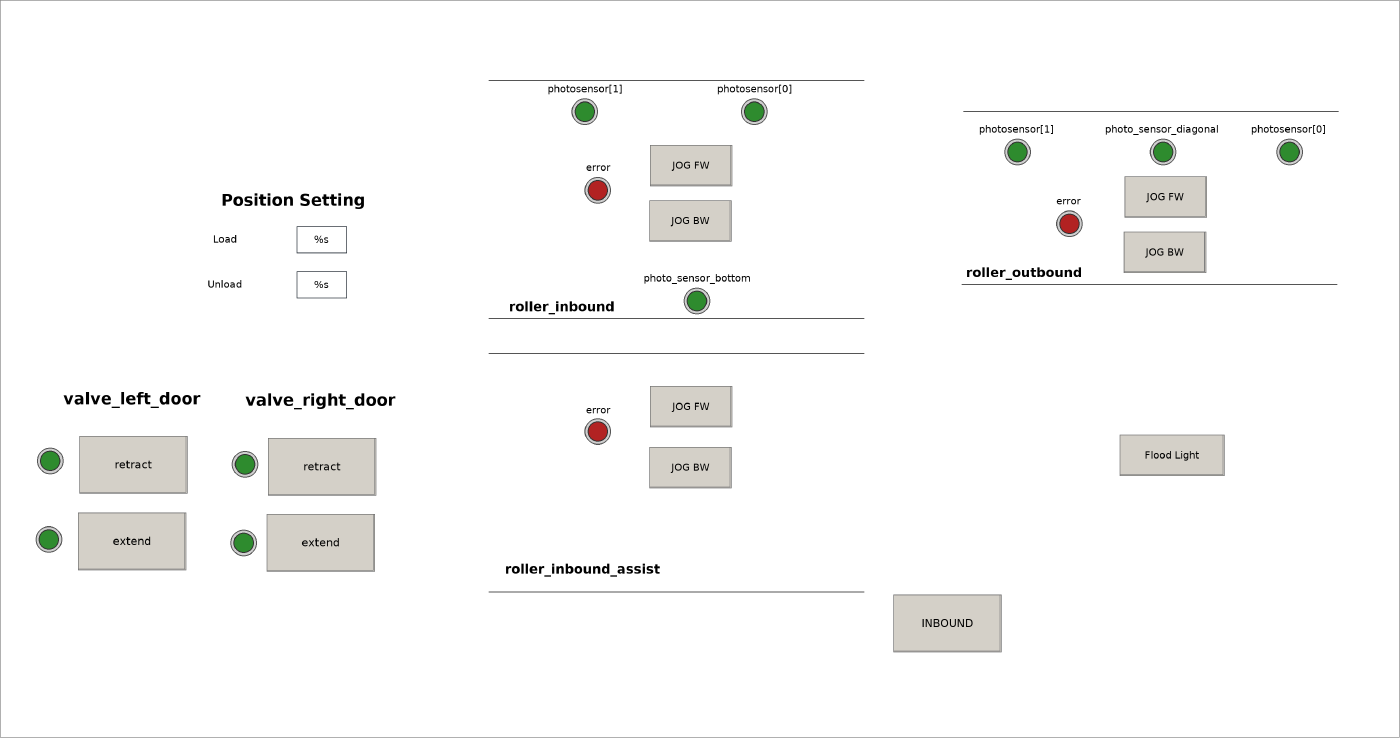
VISUALIZATION v_io_loading  // 2048x1080
    Lamp1 (1679,200 45x45), variable: GVL.fb_loading.photo_sensor_diagonal.Q, style: Lamp-Lamp1-Green
    Label (1600,176 200x26), "photo_sensor_diagonal"
    Lamp1 (1542,305 45x45), variable: GVL.fb_loading.roller_assign.roller.err.Q, style: Lamp-Lamp1-Red
    Label (1463,281 200x26), "error"
    Line (1409,163) (1958,163)
    Button (1645,258 120x60), "JOG FW", colour toggle: GVL.fb_loading.roller_assign.roller.forward
        OnMouseDown: execute { GVL.fb_loading.roller_assign.roller.forward	:= TRUE; }
        OnMouseUp: execute { GVL.fb_loading.roller_assign.roller.forward	:= FALSE; }
    Button (1644,339 120x60), "JOG BW", colour toggle: GVL.fb_loading.roller_assign.roller.backward
        OnMouseDown: execute { GVL.fb_loading.roller_assign.roller.backward	:= TRUE; }
        OnMouseUp: execute { GVL.fb_loading.roller_assign.roller.backward	:= FALSE; }
    Line (1407,416) (1956,416)
    Lamp1 (1864,200 45x45), variable: GVL.fb_loading.roller_assign.photo_sensor[0].Q, style: Lamp-Lamp1-Green
    Label (1785,176 200x26), "photosensor[0]"
    Lamp1 (1466,200 45x45), variable: GVL.fb_loading.roller_assign.photo_sensor[1].Q, style: Lamp-Lamp1-Green
    Label (1387,176 200x26), "photosensor[1]"
    Label (1398,384 200x30), "roller_outbound"
    Lamp1 (997,418 45x45), variable: GVL.fb_loading.photo_sensor_bottom.Q, style: Lamp-Lamp1-Green
    Label (920,394 200x26), "photo_sensor_bottom"
    Lamp1 (852,256 45x45), variable: GVL.fb_loading.roller_inbound.roller.err.Q, style: Lamp-Lamp1-Red
    Label (775,232 200x26), "error"
    Line (715,117) (1264,117)
    Button (951,212 120x60), "JOG FW", colour toggle: GVL.fb_loading.roller_inbound.roller.forward
        OnMouseDown: execute { GVL.fb_loading.roller_inbound.roller.forward	:= TRUE; }
        OnMouseUp: execute { GVL.fb_loading.roller_inbound.roller.forward	:= FALSE; }
    Button (950,293 120x60), "JOG BW", colour toggle: GVL.fb_loading.roller_inbound.roller.backward
        OnMouseDown: execute { GVL.fb_loading.roller_inbound.roller.backward	:= TRUE; }
        OnMouseUp: execute { GVL.fb_loading.roller_inbound.roller.backward	:= FALSE; }
    Line (715,466) (1264,466)
    Lamp1 (1081,141 45x45), variable: GVL.fb_loading.roller_inbound.photo_sensor[0].Q, style: Lamp-Lamp1-Green
    Label (1004,117 200x26), "photosensor[0]"
    Lamp1 (833,141 45x45), variable: GVL.fb_loading.roller_inbound.photo_sensor[1].Q, style: Lamp-Lamp1-Green
    Label (756,117 200x26), "photosensor[1]"
    Label (722,434 200x30), "roller_inbound"
    Button (1638,636 153x60), "Flood Light", colour toggle: GVL.fb_loading.floodlight
        toggle GVL.fb_loading.floodlight
        OnMouseDown: execute {  }
        OnMouseUp: execute {  }
    Rectangle (434,331 73x39), "%s", text variable: GVL.fb_loading.rPos_load
        OnMouseClick: write the text variable via Default, min GVL.fb_loading.rMin_lift, max GVL.fb_loading.rMax_lift
    Rectangle (434,397 73x39), "%s", text variable: GVL.fb_loading.rPos_unload
        OnMouseClick: write the text variable via Default, min GVL.fb_loading.rMin_lift, max GVL.fb_loading.rMax_lift
    Label (229,337 200x26), "Load"
    Label (229,403 200x26), "Unload"
    Label (254,280 350x26), "Position Setting"
    Lamp1 (852,609 45x45), variable: GVL.fb_loading.roller_inbound_assist.roller.err.Q, style: Lamp-Lamp1-Red
    Label (775,587 200x26), "error"
    Line (715,517) (1264,517)
    Button (951,565 120x60), "JOG FW", colour toggle: GVL.fb_loading.roller_inbound_assist.roller.forward
        OnMouseDown: execute { GVL.fb_loading.roller_inbound_assist.roller.forward	:= TRUE; }
        OnMouseUp: execute { GVL.fb_loading.roller_inbound_assist.roller.forward	:= false; }
    Button (950,654 120x60), "JOG BW", colour toggle: GVL.fb_loading.roller_inbound_assist.roller.backward
        OnMouseDown: execute { GVL.fb_loading.roller_inbound_assist.roller.backward 	:= TRUE; }
        OnMouseUp: execute { GVL.fb_loading.roller_inbound_assist.roller.backward	:= FALSE; }
    Line (715,866) (1264,866)
    Label (727,818 250x30), "roller_inbound_assist"
    Button (114,750 158x84), "extend", colour toggle: GVL.fb_loading.valve_left_door.extend
        OnMouseDown: execute { GVL.fb_loading.valve_left_door.retract := FALSE; GVL.fb_loading.valve_left_door.extend := TRUE; }
    Label (56,556 274x55), "valve_left_door"
    Button (116,638 158x84), "retract", colour toggle: GVL.fb_loading.valve_left_door.retract
        OnMouseDown: execute { GVL.fb_loading.valve_left_door.extend := FALSE; GVL.fb_loading.valve_left_door.retract := TRUE; }
    Button (390,752 158x84), "extend", colour toggle: GVL.fb_loading.valve_right_door.extend
        OnMouseDown: execute { GVL.fb_loading.valve_right_door.retract := FALSE; GVL.fb_loading.valve_right_door.extend := TRUE; }
    Label (332,558 274x55), "valve_right_door"
    Button (392,641 158x84), "retract", colour toggle: GVL.fb_loading.valve_right_door.retract
        OnMouseDown: execute { GVL.fb_loading.valve_right_door.extend := FALSE; GVL.fb_loading.valve_right_door.retract := TRUE; }
    Lamp1 (49,767 45x45), variable: GVL.fb_loading.valve_left_door.extended, style: Lamp-Lamp1-Green
    Lamp1 (51,652 45x45), variable: GVL.fb_loading.valve_left_door.retracted, style: Lamp-Lamp1-Green
    Lamp1 (334,772 45x45), variable: GVL.fb_loading.valve_right_door.extended, style: Lamp-Lamp1-Green
    Lamp1 (336,657 45x45), variable: GVL.fb_loading.valve_right_door.retracted, style: Lamp-Lamp1-Green
    Button (1307,870 158x84), "INBOUND"
        OnMouseDown: execute { GVL.fb_loading.logtech_load_status	:= LogTechTransferStatus.READY_TO_TRANSFER; }
END_VISUALIZATION

(* stored: Version 1.1.0.1, ProductVersion 3.1.4024.12
   Visu v_io_loading: Id {cd18c918-ee0d-4af8-834e-d168810db6db} *)
